# B&R Automation Studio project MappSampleProject
Automation Studio 4.2.6.110 SP; technology packages: mapp 1.50.0

## Configuration Config1

CPU X20CP1585, AutomationRuntime A4.26, Build 4.1.2, Vc V4.26.1

### Task classes (Cpu.sw)
```
Cyclic#1 (cycle 10000 us, tolerance 10000 us):
  axis01 <- MpAxisSample.axis01.prg
Cyclic#4 (cycle 100000 us, tolerance 100000 us):
  usage <- MpAxisSample.usage.prg
DataObjects: Acp10sys
NcDataObjects: acp10etxen <- acp10etxen.dob, gAxis01a <- gAxis01obj.gAxis01a.dob, gAxis01i <- gAxis01obj.gAxis01i.dob, gAxis02a <- gAxis02obj.gAxis02a.dob, gAxis02i <- gAxis02obj.gAxis02i.dob, gAxis03a <- gAxis03obj.gAxis03a.dob, gAxis03i <- gAxis03obj.gAxis03i.dob
Binaries: TCData, arsvcreg, arconfig, asfw, ashwd, iomap, User, Role, sysconf, Config, Acp10map, acp10cfg, Config_1
Libraries: MpCom, MpRecipe, sys_lib, runtime, astime, fileio, MpAxis, NcGlobal, Acp10_MC, brsystem, Acp10man, Acp10par, dataobj, powerlnk, asbrstr, asieccon
```

### Hardware
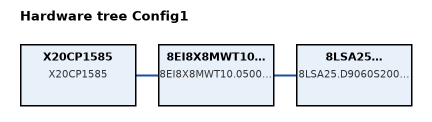
```
8EI8X8MWT10.0500-1 : 8EI8X8MWT10.0500-1 v1.0.0.3  [PLK1 -> X20CP1585.IF3 (NodeNumber=1); EC1 -> 8LSA25.D9060S200-3.EC]
  StandAloneDrive_PowerSupply = dc_powered
  DC_supply = active
  SupplyVoltage = 24
  Ax1Interface = Ax1EnDat
  Ax1DriveCtrl = Ax1OneEnc
  Ax1MPEncoder = Ax1MPEncoder1
  Ax2DriveCtrl = Ax2OneEnc
  Ax2MPEncoder = Ax2MPEncoder1
  Ax3DriveCtrl = Ax3OneEnc
  Ax3MPEncoder = Ax3MPEncoder1
8LSA25.D9060S200-3 : 8LSA25.D9060S200-3 v1.0.7.34  [EC -> 8EI8X8MWT10.0500-1.EC1; MT -> 8EI8X8MWT10.0500-1.MT1]
  MOTOR_TYPE = 16#0002
  MOTOR_COMPATIBILITY = 16#0207
  MOTOR_WIND_CONNECT = 1
  MOTOR_BRAKE_TYPE = 16#FFFF
  MOTOR_BRAKE_CURR_RATED = 0.35
  MOTOR_BRAKE_TORQ_RATED = 2.2
  MOTOR_BRAKE_ON_TIME = 0.014
  MOTOR_BRAKE_OFF_TIME = 0.028
  MOTOR_BRAKE_RESISTANCE = 0
  MOTOR_BRAKE_INDUCTANCE = 0
  MOTOR_BRAKE_VOLT_REL = 0
  MOTOR_BRAKE_VOLT_HOLD = 0
  MOTOR_BRAKE_VOLT_MAX = 0
  MOTOR_TEMPSENS_PAR1 = 31
  MOTOR_TEMPSENS_PAR2 = 289
  MOTOR_TEMPSENS_PAR3 = -30
  MOTOR_TEMPSENS_PAR4 = -0.65
  MOTOR_TEMPSENS_PAR5 = 29.06
  MOTOR_TEMPSENS_PAR6 = 58.83
  MOTOR_TEMPSENS_PAR7 = 88.17
  MOTOR_TEMPSENS_PAR8 = 117.42
  MOTOR_TEMPSENS_PAR9 = 147.14
  MOTOR_TEMPSENS_PAR10 = 175
  MOTOR_TEMPSENS_TYPE = 4353
  MOTOR_TEMPSENS_LIM = 130
  MOTOR_POLEPAIRS = 4
  MOTOR_VOLTAGE_RATED = 400
  MOTOR_VOLTAGE_CONST = 43.98
  MOTOR_SPEED_RATED = 6000
  MOTOR_SPEED_MAX = 9000
  MOTOR_TORQ_STALL = 0.6
  MOTOR_TORQ_RATED = 0.52
  MOTOR_TORQ_MAX = 2.4
  MOTOR_TORQ_CONST = 0.73
  MOTOR_CURR_STALL = 0.82
  MOTOR_CURR_RATED = 0.71
  MOTOR_CURR_MAX = 3.7
  MOTOR_WIND_CROSS_SECT = 0.055
  MOTOR_STATOR_RESISTANCE = 34.63
  MOTOR_STATOR_INDUCTANCE = 0.0496
  MOTOR_INERTIA = 2.8E-05
  MOTOR_COMMUT_OFFSET = 1000000
  MOTOR_WIND_TEMP_MAX = 110
  MOTOR_TAU_THERM = 1200
  MOTOR_AMB_TEMP_RATED = 40
  MOTOR_TEMPMODEL_REFSENS = 0
  MOTOR_TEMPMODEL_RES1 = 0
  MOTOR_TEMPMODEL_CAP1 = 0
  MOTOR_TEMPMODEL_RES2 = 0
  MOTOR_TEMPMODEL_CAP2 = 0
  MOTOR_TEMPMODEL_LOSS1 = 0
  MOTOR_TEMPMODEL_LOSS2 = 0
  MOTOR_TEMPMODEL_MODE = 16#FFFF
  MOTOR_ENCOD_TEMP_LIM = 120
X20CP1585 : X20CP1585 v1.3.0.0
  Connector IF2:
    ActivateDevice = 1
    EthInterfaceRedundant = 0
  Connector IF3:
    EplInterfaceRedundant = 0
    EplEthInterfaceRedundant = 0
  ConfigurationID = cp1382_Config1
  UserPartitionSize = 100
  TimerDeviceType = EPLX2X
  TimerDevice = X20CP1585.IF3
  TaskClassIdleTime = 10000
  Cyclic1Duration = 10000
  Cyclic1Tolerance = 10000
  Cyclic2Duration = 20000
  Cyclic2Tolerance = 20000
  Cyclic3Duration = 50000
  Cyclic3Tolerance = 50000
  Cyclic4Duration = 100000
  Cyclic4Tolerance = 100000
  Cyclic5Duration = 200000
  Cyclic5Tolerance = 200000
  Cyclic6Duration = 500000
  Cyclic6Tolerance = 500000
  Cyclic7Duration = 1000000
  Cyclic7Tolerance = 1000000
  Cyclic8Duration = 10000
  Cyclic8Tolerance = 30000000
  FileDevice1
  FileDeviceName1 = USER
  FileDevicePath1 = F:\
  FtpUser1
  FtpUsername1 = roman
  FtpUserPassword1 = 4v6oDkRIJex4249inyR9f1SYsKgW8z8c/kF9wnmvPr0=
  FtpUserSalt1 = aXUHwkaZ
  FTPAccessRight1 = 0
```

### Acp10cfg.ncc - X20CP1585/Motion/Acp10cfg.ncc
```
NcConfiguration (Version=3.14.3, NcSwId=Acp10)
  ACP10CF1_typ:
    cnt_nettrc_rec_drive = 150
    bufsize_trace_upload = 1200
    tc_nc_man_task = Cyclic #1
    glob_pv_as_ncobject = Yes
    ncsys_dl_broadcast = Yes
    ncsys_dl_acp_reset = Yes
    safemc_log_err_to_ax = Yes
    network_init:
      ncsw_init_execute = Yes
      automatic_execute = No
      node_nr_warning = Yes
      net_err_before_ncact = Yes
    nettrc:
      enter_parsecrec = Yes
      enter_ncaction = Yes
      save_ring_startidx = No
    cam_prof_download:
      cam_dat_dl_parallel = No
      tc_cam_dl_parallel = Task class for NC Manager task
    plk_if[0]:
      if_name = IF3
      tc_CycDat_PLCopen = Task class for NC Manager task
      mc_broadcast_extdat = No
```

### Acp10map.ncm - X20CP1585/Motion/Acp10map.ncm
```
NcMapping (NcSwId=Acp10)
  NcObject gAxis01 (ModuleId=8EI8X8MWT10.0500-1, Type=ncAXIS, Channel=1, AcoposSimulation=Off, InitParameter=gAxis01i, AcoposParameter=gAxis01a, Disabled=FALSE, ModuleDisabled=FALSE)
  NcObject gAxis02 (ModuleId=8EI8X8MWT10.0500-1, Type=ncAXIS, Channel=2, AcoposSimulation=Off, InitParameter=gAxis02i, AcoposParameter=gAxis02a, Disabled=FALSE, ModuleDisabled=FALSE)
  NcObject gAxis03 (ModuleId=8EI8X8MWT10.0500-1, Type=ncAXIS, Channel=3, AcoposSimulation=Off, InitParameter=gAxis03i, AcoposParameter=gAxis03a, Disabled=FALSE, ModuleDisabled=FALSE)
  NcObject 8EI8X8MWT10.0500-1_ncV_AXIS1 (ModuleId=8EI8X8MWT10.0500-1, Type=ncV_AXIS, Channel=1, Disabled=TRUE, ModuleDisabled=FALSE)
  NcObject 8EI8X8MWT10.0500-1_ncV_AXIS2 (ModuleId=8EI8X8MWT10.0500-1, Type=ncV_AXIS, Channel=2, Disabled=TRUE, ModuleDisabled=FALSE)
  NcObject 8EI8X8MWT10.0500-1_ncV_AXIS3 (ModuleId=8EI8X8MWT10.0500-1, Type=ncV_AXIS, Channel=3, Disabled=TRUE, ModuleDisabled=FALSE)
```

### Config.mprecipecsv - X20CP1585/mapp/Config.mprecipecsv
```
Element gRecipeCsv (Type=mprecipecsv)
```

### Config_1.mpaxisbasic - X20CP1585/mapp/Config_1.mpaxisbasic
```
Element gAxisBasic (Type=mpaxisbasic)
  AxisConfiguration = AxisWithConfiguration
    Drive:
      Controller:
        LoopFilters:
          [0]
          [1]
          [2]
```

## Logical view

Binary libraries used (declarations not repeated): operator, runtime, astime, AsIecCon, sys_lib, brsystem, MpCom, MpAxis, MpRecipe 1.50.0, Acp10man, Acp10par, NcGlobal, Acp10_MC

### Global.var - Global variables
```iecst
VAR
	gAxis01 : ACP10AXIS_typ;
	gAxis02 : ACP10AXIS_typ;
	gAxis03 : ACP10AXIS_typ;
END_VAR
```


### Data object Logical/acp10etxen (Ett)

- acp10etxen.ett (not shown)

### Package Logical/gAxis01obj - gAxis01obj

- Data object Logical/gAxis01obj/gAxis01a (Apt) (no source held here)

### Data object Logical/gAxis01obj/gAxis01i (Ax)

#### gAxis01i.ax
```
InitParameter (Version=3.15.1, NcSwId=ACP10)
  ACP10AXIS_typ:
    dig_in:
      level:
        reference = ncACTIV_HI
        pos_hw_end = ncACTIV_HI
        neg_hw_end = ncACTIV_HI
        trigger1 = ncACTIV_HI
        trigger2 = ncACTIV_HI
    encoder_if:
      parameter:
        count_dir = ncSTANDARD
        scaling:
          load:
            units = 36000
            rev_motor = 1
    limit:
      parameter:
        v_pos = 100000.0
        v_neg = 100000.0
        a1_pos = 500000.0
        a2_pos = 500000.0
        a1_neg = 500000.0
        a2_neg = 500000.0
        t_jolt = 0.0
        t_in_pos = 0.0
        pos_sw_end = 838860700
        neg_sw_end = -838860800
        ds_warning = 200.0
        ds_stop = 200.0
        a_stop = 1.0E+30
        dv_stop = 0.0
        dv_stop_mode = ncOFF
    controller:
      mode = ncPOSITION
      position:
        kv = 280.0
        tn = 0.0
        t_predict = 0.0004
        t_total = 0.0004
        p_max = 1.0E+30
        i_max = 1.0E+30
      speed:
        kv = 0.25
        tn = 0.0
        t_filter = 0.0
        isq_filter1:
          type = ncNOTCH
          a0 = 2358.12
          a1 = 400.0
          b0 = 0.0
          b1 = 0.0
          b2 = 0.0
          c0_par_id = 0
          c1_par_id = 0
        isq_filter2:
          type = ncOFF
          a0 = 0.0
          a1 = 0.0
          b0 = 0.0
          b1 = 0.0
          b2 = 0.0
          c0_par_id = 0
          c1_par_id = 0
        isq_filter3:
          type = ncOFF
          a0 = 0.0
          a1 = 0.0
          b0 = 0.0
          b1 = 0.0
          b2 = 0.0
          c0_par_id = 0
          c1_par_id = 0
      uf:
        type = ncLINEAR
        auto_config = ncMOTOR_PAR
        u0 = 0.0
        un = 0.0
        fn = 50.0
        k_f_slip = 0.0
      ff:
        torque_load = 0.0
        torque_pos = 0.0
        torque_neg = 0.0
        kv_torque = 0.0
        inertia = 0.0
        t_filter_a = 0.0
    move:
      stop:
        parameter[0]:
          decel_ramp = ncA_LIMIT
          controller = ncON
        parameter[1]:
          decel_ramp = ncA_LIMIT
          controller = ncON
        parameter[2]:
          decel_ramp = ncA_LIMIT
          controller = ncON
        parameter[3]:
          decel_ramp = ncA_LIMIT
          controller = ncON
        quickstop:
          decel_ramp = ncA_LIMIT
        drive_error:
          decel_ramp = ncA_LIMIT
      homing:
        parameter:
          s = 0
          v_switch = 5000.0
          v_trigger = 500.0
          a = 50000.0
          mode = ncDIRECT
          edge_sw = ncPOSITIVE
          start_dir = ncPOSITIVE
          trigg_dir = ncPOSITIVE
          ref_pulse = ncOFF
          fix_dir = ncOFF
          tr_s_block = 0.0
          torque_lim = 0.0
          ds_block = 0.0
          ds_stop = 0.0
      basis:
        parameter:
          v_pos = 10000.0
          v_neg = 10000.0
          a1_pos = 20000.0
          a2_pos = 20000.0
          a1_neg = 20000.0
          a2_neg = 20000.0
    message:
      text:
        parameter:
          format = ncBREAK
          columns = 80
          data_modul = acp10etxen
```


- Data object Logical/gAxis02obj/gAxis02a (Apt) (no source held here)

- Data object Logical/gAxis02obj/gAxis02i (Ax) (no source held here)

### Package Logical/gAxis03obj - gAxis03obj

- Data object Logical/gAxis03obj/gAxis03a (Apt) (no source held here)

### Data object Logical/gAxis03obj/gAxis03i (Ax)

#### gAxis03i.ax
```
InitParameter (Version=3.14.3, NcSwId=Acp10)
  ACP10AXIS_typ:
    dig_in:
      level:
        reference = ncACTIV_HI
        pos_hw_end = ncACTIV_LO
        neg_hw_end = ncACTIV_LO
        trigger1 = ncACTIV_HI
        trigger2 = ncACTIV_LO + ncQUICKSTOP
    encoder_if:
      parameter:
        count_dir = ncSTANDARD
        scaling:
          load:
            units = 1000
            rev_motor = 1
    limit:
      parameter:
        v_pos = 10000
        v_neg = 10000
        a1_pos = 50000
        a2_pos = 50000
        a1_neg = 50000
        a2_neg = 50000
        t_jolt = 0
        t_in_pos = 0
        pos_sw_end = 2000000000
        neg_sw_end = -2000000000
        ds_warning = 500
        ds_stop = 1000
        a_stop = 1.0e30
        dv_stop = 0
        dv_stop_mode = ncOFF
    controller:
      mode = ncPOSITION
      position:
        kv = 50
        tn = 0
        t_predict = 0.0004
        t_total = 0.0004
        p_max = 1.0e30
        i_max = 0
      speed:
        kv = 2.0
        tn = 0
        t_filter = 0.0
        isq_filter1:
          type = ncOFF
          a0 = 0.0
          a1 = 0.0
          b0 = 0.0
          b1 = 0.0
          b2 = 0.0
          c0_par_id = 0
          c1_par_id = 0
        isq_filter2:
          type = ncOFF
          a0 = 0.0
          a1 = 0.0
          b0 = 0.0
          b1 = 0.0
          b2 = 0.0
          c0_par_id = 0
          c1_par_id = 0
        isq_filter3:
          type = ncOFF
          a0 = 0.0
          a1 = 0.0
          b0 = 0.0
          b1 = 0.0
          b2 = 0.0
          c0_par_id = 0
          c1_par_id = 0
      uf:
        type = ncLINEAR
        auto_config = ncMOTOR_PAR
        u0 = 0
        un = 0
        fn = 50.0
        k_f_slip = 0
      ff:
        torque_load = 0.0
        torque_pos = 0.0
        torque_neg = 0.0
        kv_torque = 0.0
        inertia = 0.0
        t_filter_a = 0.0
    move:
      stop:
        parameter[0]:
          decel_ramp = ncA_LIMIT
          controller = ncON
        parameter[1]:
          decel_ramp = ncA_LIMIT
          controller = ncON
        parameter[2]:
          decel_ramp = ncA_LIMIT
          controller = ncON
        parameter[3]:
          decel_ramp = ncA_LIMIT
          controller = ncON
        quickstop:
          decel_ramp = ncA_LIMIT
        drive_error:
          decel_ramp = ncA_LIMIT
      homing:
        parameter:
          s = 0
          v_switch = 5000
          v_trigger = 500
          a = 50000
          mode = ncDIRECT
          edge_sw = ncPOSITIVE
          start_dir = ncPOSITIVE
          trigg_dir = ncPOSITIVE
          ref_pulse = ncOFF
          fix_dir = ncOFF
          tr_s_block = 0
          torque_lim = 0
          ds_block = 0
          ds_stop = 0
      basis:
        parameter:
          v_pos = 5000
          v_neg = 5000
          a1_pos = 50000
          a2_pos = 50000
          a1_neg = 50000
          a2_neg = 50000
    message:
      text:
        parameter:
          format = ncBREAK
          columns = 80
          data_modul = acp10etxen
```

Listed in the project but not available here: Logical/Global.typ, Logical/MpRecipeSample, Logical/MpAxisSample
